FUNCTION_BLOCK fb_ratio_trimming

VAR_INPUT
	loop14: REAL;
	loop15: REAL;
END_VAR

VAR_OUTPUT
	r1: REAL := 0.0;
	r4: REAL := 0.0;
END_VAR

VAR
END_VAR


r1 := loop14 + r1;
r4 := loop15 - loop14 + r4;

END_FUNCTION_BLOCK

(* stored: Version 1.1.0.1, ProductVersion 3.1.0.26
   POU fb_ratio_trimming: Id {d3cfa3b6-537a-4da3-a8d7-0f48afbd3e17} *)
